// TIA Portal V20 export
TYPE "LER_typeSequenceRelation"
// stored: Access Published
   STRUCT
      homeCheck { ExternalWritable := 'False'} : Array[0..99] of Bool;   // Check The Status Of Each Homing
      selectJobStatus { ExternalWritable := 'False'} : Array[0..99] of "LAF_typeJobStatus";
      JobInterface { ExternalWritable := 'False'} : "LER_typeJobInterface";   // Interface To Check Equipment Modules Status
   END_STRUCT;
END_TYPE
